FUNCTION_BLOCK TertFiltPumpMgr (* Basic Function Block Type *)
  (* Standard: 61499-2 *)
  (* Version 0.0, 12/17/2025, SESA313294, Schneider Electric, Template *)
  PACKAGE SE.Nereda;
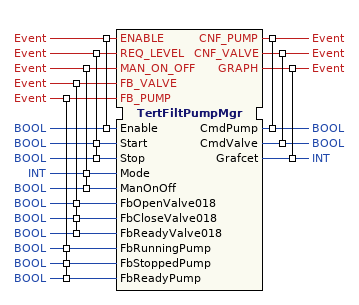
  EVENT_INPUT
    ENABLE WITH Enable;
    REQ_LEVEL WITH Start, Stop; (* Normal Execution Request *)
    MAN_ON_OFF WITH ManOnOff, Mode;
    FB_VALVE WITH FbOpenValve018, FbCloseValve018, FbReadyValve018;
    FB_PUMP WITH FbRunningPump, FbStoppedPump, FbReadyPump;
  END_EVENT
  EVENT_OUTPUT
    CNF_PUMP WITH CmdPump;
    CNF_VALVE WITH CmdValve;
    GRAPH WITH Grafcet;
  END_EVENT
  VAR_INPUT
    Enable : BOOL;
    Start : BOOL;
    Stop : BOOL;
    Mode : INT;
    ManOnOff : BOOL;
    FbOpenValve018 : BOOL;
    FbCloseValve018 : BOOL;
    FbReadyValve018 : BOOL;
    FbRunningPump : BOOL;
    FbStoppedPump : BOOL;
    FbReadyPump : BOOL;
  END_VAR
  VAR_OUTPUT
    CmdPump : BOOL;
    CmdValve : BOOL;
    Grafcet : INT;
  END_VAR
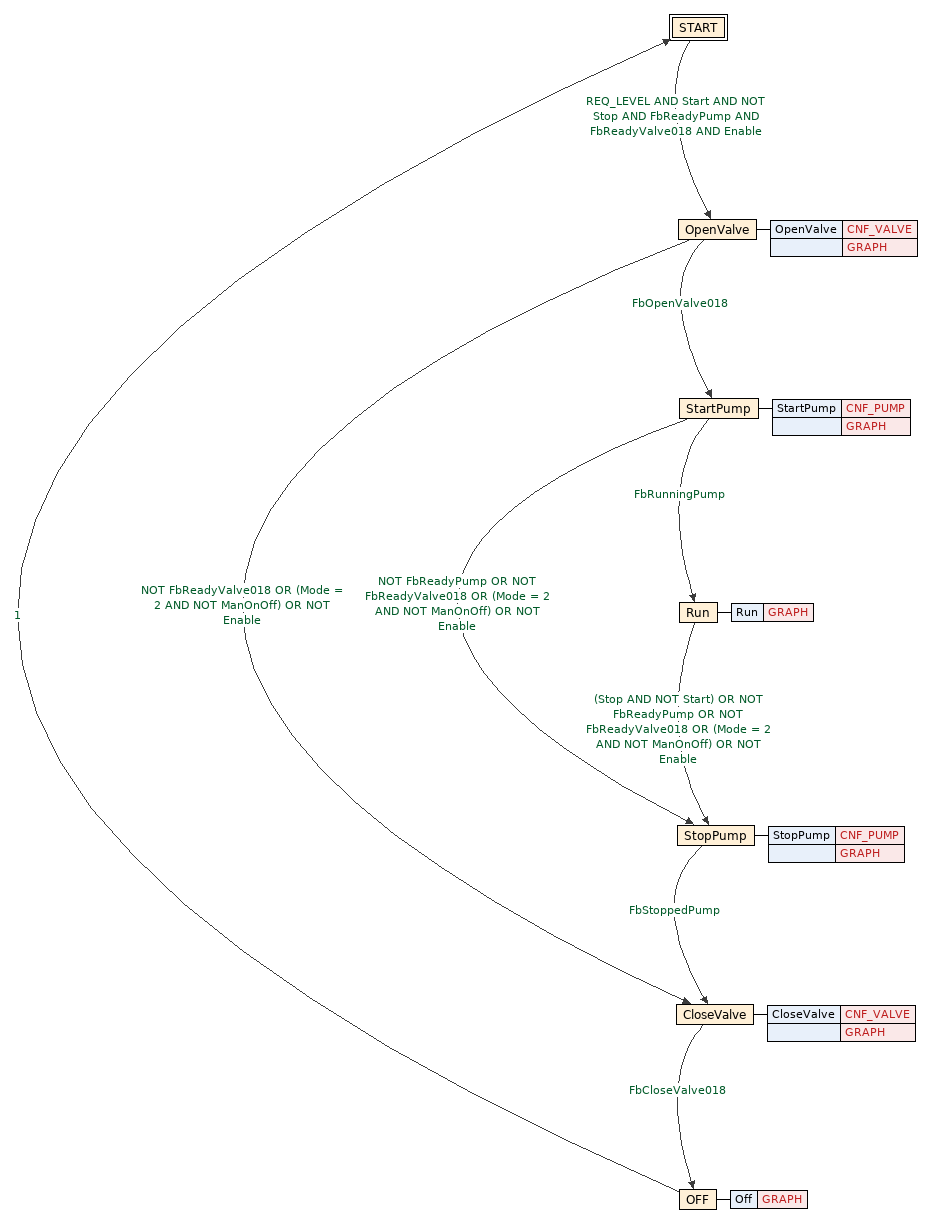
  EC_STATES
    START; (* Initial State *)
    OpenValve : OpenValve -> CNF_VALVE, -> GRAPH;
    StartPump : StartPump -> CNF_PUMP, -> GRAPH;
    Run : Run -> GRAPH;
    CloseValve : CloseValve -> CNF_VALVE, -> GRAPH;
    StopPump : StopPump -> CNF_PUMP, -> GRAPH;
    OFF : Off -> GRAPH;
  END_STATES
  EC_TRANSITIONS
    StopPump TO CloseValve := FbStoppedPump;
    START TO OpenValve := REQ_LEVEL AND Start AND NOT Stop AND FbReadyPump AND FbReadyValve018 AND Enable;
    OpenValve TO StartPump := FbOpenValve018;
    StartPump TO Run := FbRunningPump;
    Run TO StopPump := (Stop AND NOT Start) OR NOT FbReadyPump OR NOT FbReadyValve018 OR (Mode = 2 AND NOT ManOnOff) OR NOT Enable;
    OFF TO START := 1;
    OpenValve TO CloseValve := NOT FbReadyValve018 OR (Mode = 2 AND NOT ManOnOff) OR NOT Enable;
    StartPump TO StopPump := NOT FbReadyPump OR NOT FbReadyValve018 OR (Mode = 2 AND NOT ManOnOff) OR NOT Enable;
    CloseValve TO OFF := FbCloseValve018;
  END_TRANSITIONS
  ALGORITHM OpenValve IN ST:
CmdValve := TRUE;
Grafcet := 1;
  END_ALGORITHM
  ALGORITHM StartPump IN ST:
CmdPump := TRUE;
Grafcet := 2;
  END_ALGORITHM
  ALGORITHM StopPump IN ST:
CmdPump := FALSE;
Grafcet := 4;
  END_ALGORITHM
  ALGORITHM CloseValve IN ST:
CmdValve := FALSE;
Grafcet := 5;
  END_ALGORITHM
  ALGORITHM Run IN ST:
;
Grafcet := 3;
  END_ALGORITHM
  ALGORITHM Off IN ST:
;
Grafcet := 6;
  END_ALGORITHM
END_FUNCTION_BLOCK
